VAR_GLOBAL
	CTC_MOTION_MODE_OFF 		:USINT := 0;
	CTC_MOTION_MODE_HALT 		:USINT := 1;
	CTC_MOTION_MODE_TEACH 		:USINT := 2;
	CTC_MOTION_MODE_MOVEOUT 	:USINT := 3;
	CTC_MOTION_MODE_MOVEIN 		:USINT := 4;
	CTC_MOTION_MODE_FREEPOS 	:USINT := 5;
	CTC_MOTION_MODE_FREEPOSPRO 	:USINT := 6;
	CTC_MOTION_MODE_HOME 		:USINT := 7;
	CTC_MOTION_MODE_RESET 		:USINT := 255;
	CTC_MOTION_MODE_FREEPOSREL 	:USINT := 30;
	CTC_MOTION_MODE_FREEVEL 	:USINT := 31;
	CTC_MOTION_MODE_FREETORQUE 	:USINT := 32;
	CTC_MOTION_MODE_DONOTHING	:USINT := 128;
	//	
	CTC_STATUS_BYTE_IDLE 		:USINT := 0;
	CTC_STATUS_BYTE_READY 		:USINT := 1;
	CTC_STATUS_BYTE_ACTIVE 		:USINT := 2;
	CTC_STATUS_BYTE_ERROR 		:USINT := 3;
	CTC_STATUS_BYTE_TEACH 		:USINT := 4;
END_VAR

(* stored: Version 1.1.0.1, ProductVersion 3.1.4026.17
   GVL CTC_CONSTANTS: Id {69143ece-bf22-469f-a3c9-e861e84f9dfc} *)
